{attribute 'qualified_only'}
VAR_GLOBAL PERSISTENT
		PCB_Batch_ID			: INT;


END_VAR

(* stored: Version 1.1.0.1, ProductVersion 3.1.4024.3
   GVL GVL_Persistent: Id {1c3e328e-f603-4a6c-b1ff-033918966c31} *)
